TYPE typ_FBInt_Debounce :
STRUCT
	I		: typFBDInput;
	IQ		: typFBDInOut;
	Q		: typFBDOutput;
END_STRUCT
END_TYPE

(* stored: Version 1.1.0.1, ProductVersion 3.1.4024.6
   DUT typ_FBInt_Debounce: Id {0dafd016-cddd-4755-8d94-a3e036095308} *)
